FUNCTION_BLOCK Axis_Move
VAR_INPUT
	Input1:BOOL;
END_VAR
VAR_OUTPUT
END_VAR
VAR
	absMove1: MC_MoveAbsolute;
	absMove2: MC_MoveAbsolute;
	pulse1:R_TRIG;
	Pulse2:R_TRIG;
	Pulse3:R_TRIG;
	CTU1:CTU;
	AxisStop:MC_Stop;
	trig1: F_TRIG;

END_VAR

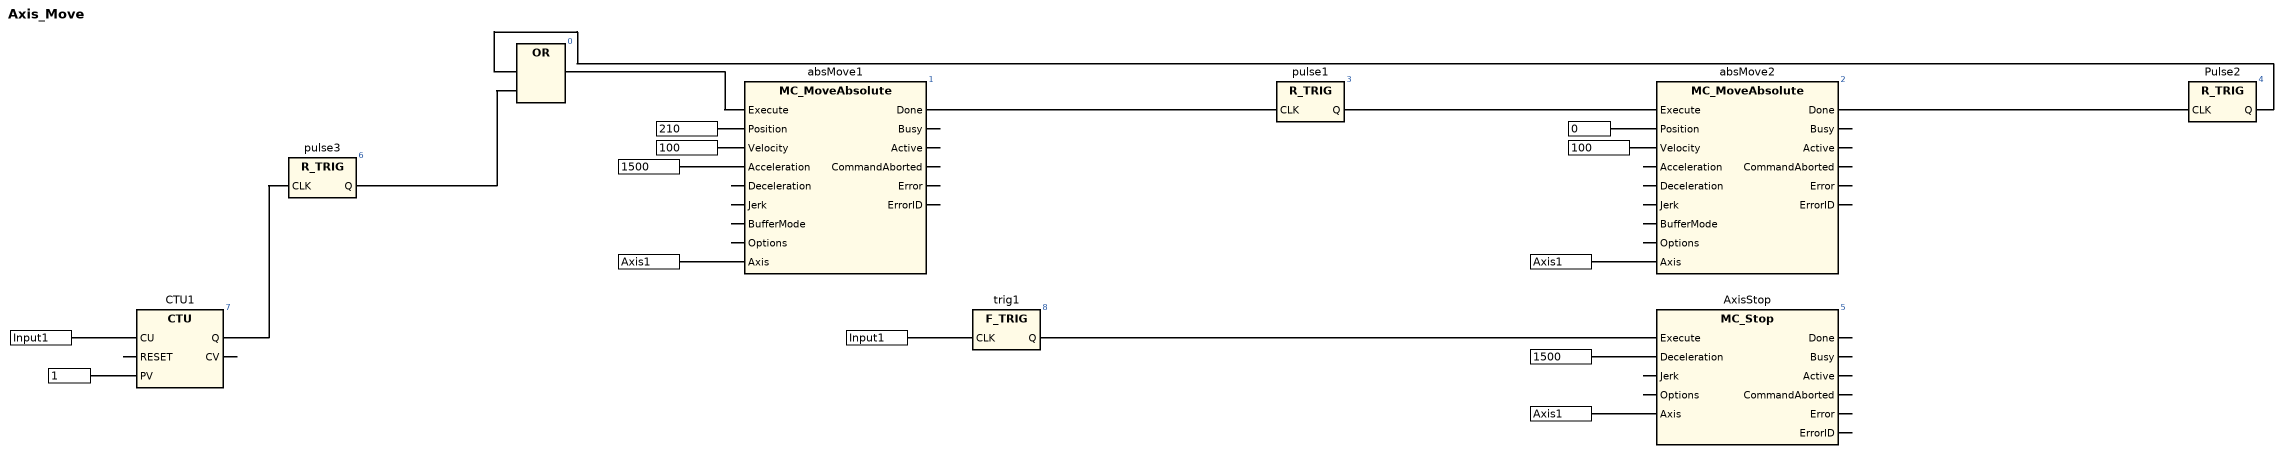
absMove1(
    Execute := Pulse2.Q OR pulse3.Q,
    Position := 210,
    Velocity := 100,
    Acceleration := 1500,
    Axis := Axis1); // MC_MoveAbsolute
absMove2(Execute := pulse1.Q, Position := 0, Velocity := 100, Axis := Axis1); // MC_MoveAbsolute
pulse1(CLK := absMove1.Done); // R_TRIG
Pulse2(CLK := absMove2.Done); // R_TRIG
AxisStop(Execute := trig1.Q, Deceleration := 1500, Axis := Axis1); // MC_Stop
pulse3(CLK := CTU1.Q); // R_TRIG
CTU1(CU := Input1, PV := 1); // CTU
trig1(CLK := Input1); // F_TRIG

END_FUNCTION_BLOCK

(* stored: Version 1.1.0.1, ProductVersion 3.1.4024.12
   POU Axis_Move: Id {4ecd53e7-77fd-44aa-abfa-d3954ba81ce2}, SpecialFunc None *)
